{attribute 'to_string'}
TYPE Pushbutton_Enum :
(
	PB_EStop	:= 0,
	PB_Start	:= 1,
	PB_Stop		:= 2,
	PB_Reset	:= 3
);
END_TYPE

(* stored: Version 1.1.0.1
   DUT Pushbutton_Enum: Id {fdf8b117-916e-439c-8a30-699e1501f821} *)
